Staubli VAL3: _PA_grd_fin.dtx

mdesc mNomSpeed = {tmax=25, rmax=25, blend=off}
bool bRunning
num nLastCmd
num nStatusSignal
num nWaypointCount
num nConnFlag
bool bMove
bool bAlterRun
num nAlterBegin
num nAlter
num nAlterEnd
public sio siTcpIpCommand = {link=Socket\Command}
public sio siTcpIpMotion = {link=Socket\Motion}
public sio siTcpIpFbk = {link=Socket\Feedback}
jointRx jHome = {j1=81.48, j2=37.87, j3=86.46, j4=-16.98, j5=-30.36, j6=14}
tool tTool = {x=225.4998, y=-0.0005, z=145.3992, ry=-90, fatherId=flange[0], ioLink=valve1}
mdesc mAlterspeed = {tmax=500, rmax=500}
trsf trOffset
public aio aiECAT1_0 = {link=EtherCAT-1\%IF0}
public dio doECAT1_192 = {link=EtherCAT-1\%Q192}
public aio aoECAT1_0 = {link=EtherCAT-1\%QF0}
public aio aoECAT1_32 = {link=EtherCAT-1\%QF32}
public aio aoECAT1_64 = {link=EtherCAT-1\%QF64}
public aio aoECAT1_96 = {link=EtherCAT-1\%QF96}
public aio aoECAT1_128 = {link=EtherCAT-1\%QF128}
public aio aoECAT1_160 = {link=EtherCAT-1\%QF160}
pointRx pCurent_pos = {fatherId=world[0]}
bool bAlterReset
num nDeltZ
num l_nHeight
pointRx pStart = {fatherId=world[0]}
pointRx pEnd = {fatherId=world[0]}
pointRx pApproach = {fatherId=world[0]}
pointRx pRetract = {fatherId=world[0]}
pointRx pWaypoints[100]
  [0] = {fatherId=world[0]}
  [1] = {fatherId=world[0]}
  [2] = {fatherId=world[0]}
  [3] = {fatherId=world[0]}
  [4] = {fatherId=world[0]}
  [5] = {fatherId=world[0]}
  [6] = {fatherId=world[0]}
  [7] = {fatherId=world[0]}
  [8] = {fatherId=world[0]}
  [9] = {fatherId=world[0]}
  [10] = {fatherId=world[0]}
  [11] = {fatherId=world[0]}
  [12] = {fatherId=world[0]}
  [13] = {fatherId=world[0]}
  [14] = {fatherId=world[0]}
  [15] = {fatherId=world[0]}
  [16] = {fatherId=world[0]}
  [17] = {fatherId=world[0]}
  [18] = {fatherId=world[0]}
  [19] = {fatherId=world[0]}
  [20] = {fatherId=world[0]}
  [21] = {fatherId=world[0]}
  [22] = {fatherId=world[0]}
  [23] = {fatherId=world[0]}
  [24] = {fatherId=world[0]}
  [25] = {fatherId=world[0]}
  [26] = {fatherId=world[0]}
  [27] = {fatherId=world[0]}
  [28] = {fatherId=world[0]}
  [29] = {fatherId=world[0]}
  [30] = {fatherId=world[0]}
  [31] = {fatherId=world[0]}
  [32] = {fatherId=world[0]}
  [33] = {fatherId=world[0]}
  [34] = {fatherId=world[0]}
  [35] = {fatherId=world[0]}
  [36] = {fatherId=world[0]}
  [37] = {fatherId=world[0]}
  [38] = {fatherId=world[0]}
  [39] = {fatherId=world[0]}
  [40] = {fatherId=world[0]}
  [41] = {fatherId=world[0]}
  [42] = {fatherId=world[0]}
  [43] = {fatherId=world[0]}
  [44] = {fatherId=world[0]}
  [45] = {fatherId=world[0]}
  [46] = {fatherId=world[0]}
  [47] = {fatherId=world[0]}
  [48] = {fatherId=world[0]}
  [49] = {fatherId=world[0]}
  [50] = {fatherId=world[0]}
  [51] = {fatherId=world[0]}
  [52] = {fatherId=world[0]}
  [53] = {fatherId=world[0]}
  [54] = {fatherId=world[0]}
  [55] = {fatherId=world[0]}
  [56] = {fatherId=world[0]}
  [57] = {fatherId=world[0]}
  [58] = {fatherId=world[0]}
  [59] = {fatherId=world[0]}
  [60] = {fatherId=world[0]}
  [61] = {fatherId=world[0]}
  [62] = {fatherId=world[0]}
  [63] = {fatherId=world[0]}
  [64] = {fatherId=world[0]}
  [65] = {fatherId=world[0]}
  [66] = {fatherId=world[0]}
  [67] = {fatherId=world[0]}
  [68] = {fatherId=world[0]}
  [69] = {fatherId=world[0]}
  [70] = {fatherId=world[0]}
  [71] = {fatherId=world[0]}
  [72] = {fatherId=world[0]}
  [73] = {fatherId=world[0]}
  [74] = {fatherId=world[0]}
  [75] = {fatherId=world[0]}
  [76] = {fatherId=world[0]}
  [77] = {fatherId=world[0]}
  [78] = {fatherId=world[0]}
  [79] = {fatherId=world[0]}
  [80] = {fatherId=world[0]}
  [81] = {fatherId=world[0]}
  [82] = {fatherId=world[0]}
  [83] = {fatherId=world[0]}
  [84] = {fatherId=world[0]}
  [85] = {fatherId=world[0]}
  [86] = {fatherId=world[0]}
  [87] = {fatherId=world[0]}
  [88] = {fatherId=world[0]}
  [89] = {fatherId=world[0]}
  [90] = {fatherId=world[0]}
  [91] = {fatherId=world[0]}
  [92] = {fatherId=world[0]}
  [93] = {fatherId=world[0]}
  [94] = {fatherId=world[0]}
  [95] = {fatherId=world[0]}
  [96] = {fatherId=world[0]}
  [97] = {fatherId=world[0]}
  [98] = {fatherId=world[0]}
  [99] = {fatherId=world[0]}
mdesc mAprSpeed = {tmax=10, rmax=10}
num i
mdesc mGrindSpeed = {tmax=10, rmax=10}
jointRx jScan = {j1=83.61, j2=38.15, j3=96.24, j4=-4.09, j5=-58.18, j6=-4.12}
num nByte
num nCmdSignal
num nForceTarget
num nX
num nY
num nZ
num nRx
num nRy
num nRz
num nKey
num x_nValue
public sio siTcpIpJoint = {link=Socket\Joint}
jointRx jCurrent
string l_sData
